{attribute 'GeneratedUsingTerminal: IODEVICETYPE_ETHERCATPROT'}
{attribute addProperty BoxType "IODEVICETYPE_ETHERCATPROT"}
{attribute addProperty Id "Term_9_EK1100Term_9_EK1100_91BFEC251351SyncUnitsSyncUnits_732A48E445InputsInputs_A65FACA410OutputsOutputs_23C0ED1D6InfoDataInfoData_84133AC922"}
{attribute addProperty CRC "494125692"}
{attribute addProperty Size "1434"}
{attribute addProperty Name "Device 4 (EtherCAT)"}
TYPE Device_4_EtherCAT_1D73C27C EXTENDS TcoIo.EtcMasterBase_62654B43 :
STRUCT
	{attribute addProperty Name "Term 9 (EK1100)"}
	{attribute addProperty PreviousPort "Device 4 (EtherCAT) : Master"}
	Term_9_EK1100 : Term_9_EK1100_91BFEC25;
	{attribute addProperty Name "SyncUnits"}
	SyncUnits : SyncUnits_732A48E4;
	{attribute addProperty Name "Inputs"}
	Inputs : TcoIo.Inputs_A65FACA4;
	{attribute addProperty Name "Outputs"}
	Outputs : TcoIo.Outputs_23C0ED1D;
	{attribute addProperty Name "InfoData"}
	InfoData : TcoIo.InfoData_84133AC9;
END_STRUCT
END_TYPE

(* stored: Version 1.2.0.0, ProductVersion 3.1.4024.11
   DUT Device_4_EtherCAT_1D73C27C: Id {8847703d-a196-038e-1f5f-34c1d37d03fe} *)
